// TIA Portal V20 export
DATA_BLOCK "FDI1"   // DB292
// stored: MemoryReserve 100
   VAR
      "MANIFOLD-1 SOL POWER MC FEEDBACK" : Bool;
      "MANIFOLD-2 SOL POWER MC FEEDBACK" : Bool;
      SPARE1 : Bool;
      SPARE2 : Bool;
      "FFU POWER MC 1 FEEDBACK" : Bool;
      "FFU POWER MC 2 FEEDBACK" : Bool;
      SPARE3 : Bool;
      SPARE4 : Bool;
   END_VAR
BEGIN
END_DATA_BLOCK
